// TIA Portal V19 export
TYPE "UDT_Auftrag_Pos"
   STRUCT
      Fertig : Bool;
      Abholbar : Bool;
      Sperre : Bool;
      CheckSperre : Bool;
      WT_151 : Bool;
      Wt_Typ : Byte;
      Wt_Cmd : Byte;
      Oldest : Real;
   END_STRUCT;
END_TYPE
